// TwinCAT 3 PLC project FMMathTests
// ProgramVersion: 3.1.4024.0
// libraries:
//   Math, * (TomasRompotl)
//   Tc3_Module, * (Beckhoff Automation GmbH)
//   TcUnit, * (www.tcunit.org)
// project tree:
//   / PlcTask.TcTTO (not stored), PRG_Test.TcPOU
//   Range/ IsInRangeInclusiveFunctionsTest.TcPOU
// (motion and I/O tree: see PLC project fmtypestests)
// real-time tasks:
//   TASK FMTypesTestsTask: cycle T#1ms, priority 20, ADS port 350
//   TASK FMStringsTestsTask: cycle T#1ms, priority 21, ADS port 351
//   TASK FMDataTestsTask: cycle T#1ms, priority 22, ADS port 352
//   TASK FMMathTestsTask: cycle T#1ms, priority 23, ADS port 353
//   TASK FMTimeTestsTask: cycle T#1ms, priority 24, ADS port 354

// ---- PRG_Test.TcPOU
PROGRAM PRG_Test
VAR
	isInRangeFunctionsTest : IsInRangeInclusiveFunctionsTest;
END_VAR

TcUnit.RUN();

END_PROGRAM

// ---- Range/IsInRangeInclusiveFunctionsTest.TcPOU
FUNCTION_BLOCK IsInRangeInclusiveFunctionsTest EXTENDS FB_TestSuite
VAR
END_VAR

IsInRangeInclusiveFunction();
IsInRangeInclusive2DFunction();
IsInRangeInclusive3DFunction();

METHOD IsInRangeInclusive2DFunction
VAR
	point : Point2D;
	range : Range2D;
END_VAR
TcUnit.TEST('IsInRangeInclusive2D tests');

// Point inside range (nominal)
point.X := 5;
point.Y := 5;
range.X.Bottom := 0;
range.X.Top := 10;
range.Y.Bottom := 0;
range.Y.Top := 10;
AssertEquals_BOOL(
	Expected := TRUE,
	Actual := IsInRangeInclusive2D(point, range),
	Message := 'Point inside 2D range should return TRUE');

// Point on boundary
point.X := 0;
point.Y := 10;
range.X.Bottom := 0;
range.X.Top := 10;
range.Y.Bottom := 0;
range.Y.Top := 10;
AssertEquals_BOOL(
	Expected := TRUE,
	Actual := IsInRangeInclusive2D(point, range),
	Message := 'Point on boundary should return TRUE');

// Point outside in one dimension
point.X := 5;
point.Y := 11;
range.X.Bottom := 0;
range.X.Top := 10;
range.Y.Bottom := 0;
range.Y.Top := 10;
AssertEquals_BOOL(
	Expected := FALSE,
	Actual := IsInRangeInclusive2D(point, range),
	Message := 'Point outside one dimension should return FALSE');

// Invalid range in one dimension
point.X := 5;
point.Y := 5;
range.X.Bottom := 10;
range.X.Top := 0;
range.Y.Bottom := 0;
range.Y.Top := 10;
AssertEquals_BOOL(
	Expected := FALSE,
	Actual := IsInRangeInclusive2D(point, range),
	Message := 'Invalid range in one dimension should return FALSE');

TEST_FINISHED();
END_METHOD

METHOD IsInRangeInclusive3DFunction
VAR
	point : Point3D;
	range : Range3D;
END_VAR
TcUnit.TEST('IsInRangeInclusive3D tests');

// Point inside range (nominal)
point.X := 5;
point.Y := 5;
point.Z := 5;
range.X.Bottom := 0;
range.X.Top := 10;
range.Y.Bottom := 0;
range.Y.Top := 10;
range.Z.Bottom := 0;
range.Z.Top := 10;
AssertEquals_BOOL(
	Expected := TRUE,
	Actual := IsInRangeInclusive3D(point, range),
	Message := 'Point inside 3D range should return TRUE');

// Point on boundary
point.X := 0;
point.Y := 10;
point.Z := 0;
range.X.Bottom := 0;
range.X.Top := 10;
range.Y.Bottom := 0;
range.Y.Top := 10;
range.Z.Bottom := 0;
range.Z.Top := 10;
AssertEquals_BOOL(
	Expected := TRUE,
	Actual := IsInRangeInclusive3D(point, range),
	Message := 'Point on boundary should return TRUE');

// Point outside in one dimension
point.X := 5;
point.Y := 5;
point.Z := 11;
range.X.Bottom := 0;
range.X.Top := 10;
range.Y.Bottom := 0;
range.Y.Top := 10;
range.Z.Bottom := 0;
range.Z.Top := 10;
AssertEquals_BOOL(
	Expected := FALSE,
	Actual := IsInRangeInclusive3D(point, range),
	Message := 'Point outside one dimension should return FALSE');

// Invalid range in one dimension
point.X := 5;
point.Y := 5;
point.Z := 5;
range.X.Bottom := 10;
range.X.Top := 0;
range.Y.Bottom := 0;
range.Y.Top := 10;
range.Z.Bottom := 0;
range.Z.Top := 10;
AssertEquals_BOOL(
	Expected := FALSE,
	Actual := IsInRangeInclusive3D(point, range),
	Message := 'Invalid range in one dimension should return FALSE');

TEST_FINISHED();
END_METHOD

METHOD IsInRangeInclusiveFunction
VAR
	range : Range;
END_VAR
TcUnit.TEST('IsInRangeInclusive tests');

// Value inside range
range.Bottom := 0;
range.Top := 10;
AssertEquals_BOOL(
	Expected := TRUE,
	Actual := IsInRangeInclusive(5, range),
	Message := 'Value inside range should return TRUE');

// Value equal to Bottom
range.Bottom := 0;
range.Top := 10;
AssertEquals_BOOL(
	Expected := TRUE,
	Actual := IsInRangeInclusive(0, range),
	Message := 'Value equal to Bottom should return TRUE');

// Value equal to Top
range.Bottom := 0;
range.Top := 10;
AssertEquals_BOOL(
	Expected := TRUE,
	Actual := IsInRangeInclusive(10, range),
	Message := 'Value equal to Top should return TRUE');

// Value below Bottom
range.Bottom := 0;
range.Top := 10;
AssertEquals_BOOL(
	Expected := FALSE,
	Actual := IsInRangeInclusive(-1, range),
	Message := 'Value below Bottom should return FALSE');

// Value above Top
range.Bottom := 0;
range.Top := 10;
AssertEquals_BOOL(
	Expected := FALSE,
	Actual := IsInRangeInclusive(11, range),
	Message := 'Value above Top should return FALSE');

// Invalid range (Bottom > Top)
range.Bottom := 10;
range.Top := 0;
AssertEquals_BOOL(
	Expected := FALSE,
	Actual := IsInRangeInclusive(5, range),
	Message := 'Invalid range (Bottom > Top) should return FALSE');

// Zero-width range (Bottom = Top), value matches
range.Bottom := 0;
range.Top := 0;
AssertEquals_BOOL(
	Expected := TRUE,
	Actual := IsInRangeInclusive(0, range),
	Message := 'Value equal to zero-range should return TRUE');

// Zero-width range (Bottom = Top), value does not match
range.Bottom := 0;
range.Top := 0;
AssertEquals_BOOL(
	Expected := FALSE,
	Actual := IsInRangeInclusive(0.1, range),
	Message := 'Value outside zero-range should return FALSE');

TEST_FINISHED();
END_METHOD

END_FUNCTION_BLOCK
